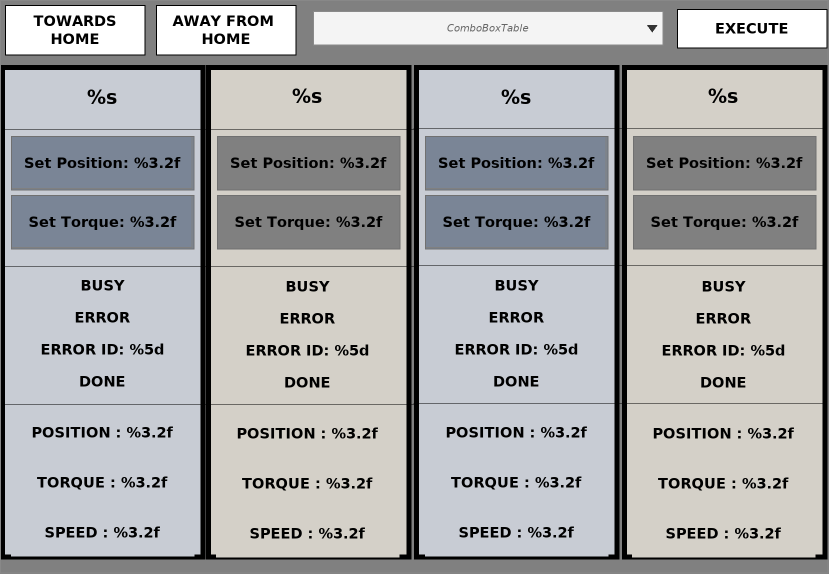
VISUALIZATION motorControlScreen  // 829x574
    Rectangle (206,65 205x494)
    RoundedRectangle (677,9 150x39), "EXECUTE", colour toggle: multiControl.bExecute
        toggle multiControl.bExecute
    ComboBoxTable (313,11 350x34), variable: multiControl.nActionIndex, data array: multiControl.aActionList
        p3854506369: multiControl.aActionList[INDEX]
    Rectangle (0,65 205x494)
    Rectangle (414,65 205x494)
    Rectangle (622,65 205x494)
    RoundedRectangle (10,71 185x53), "%s", text variable: multiControl.sMotorDisp1, colour toggle: multiControl.aMotorEnable[1]
        p55702900: multiControl.aDispFontColor[1]
        toggle multiControl.aMotorEnable[1]
    Rectangle (11,409 183x47), "POSITION : %3.2f", text variable: multiControl.aMotorPos[1]
    Rectangle (11,271 183x29), "BUSY", colour toggle: multiControl.aMotorBusy[1]
    Rectangle (11,367 183x29), "DONE", colour toggle: multiControl.aMotorDone[1]
    Rectangle (11,303 183x29), "ERROR", colour toggle: multiControl.aMotorError[1]
    Rectangle (11,335 183x29), "ERROR ID: %5d", text variable: multiControl.aMotorErrorId[1]
    Rectangle (11,459 183x47), "TORQUE : %3.2f", text variable: multiControl.aMotorTorque[1]
    Rectangle (11,509 183x47), "SPEED : %3.2f", text variable: multiControl.aMotorSpeed[1]
    Button (11,136 183x54), "Set Position: %3.2f", text variable: multiControl.aMotorSetPos[1]
        OnMouseClick: write the text variable via VisuDialogs.Numpad
    Button (11,195 183x54), "Set Torque: %3.2f", text variable: multiControl.aMotorSetTorq[1]
        OnMouseClick: write the text variable via VisuDialogs.Numpad
    Line (0,129) (827,128)
    Line (1,266) (828,265)
    Line (0,404) (827,403)
    Button (217,195 183x54), "Set Torque: %3.2f", text variable: multiControl.aMotorSetTorq[2]
        OnMouseClick: write the text variable via VisuDialogs.Numpad
    Button (217,136 183x54), "Set Position: %3.2f", text variable: multiControl.aMotorSetPos[2]
        OnMouseClick: write the text variable via VisuDialogs.Numpad
    RoundedRectangle (215,70 185x53), "%s", text variable: multiControl.sMotorDisp2, colour toggle: multiControl.aMotorEnable[2]
        p55702900: multiControl.aDispFontColor[2]
        toggle multiControl.aMotorEnable[2]
    Rectangle (216,272 183x29), "BUSY", colour toggle: multiControl.aMotorBusy[2]
    Rectangle (216,410 183x47), "POSITION : %3.2f", text variable: multiControl.aMotorPos[2]
    Rectangle (216,368 183x29), "DONE", colour toggle: multiControl.aMotorDone[2]
    Rectangle (216,304 183x29), "ERROR", colour toggle: multiControl.aMotorError[2]
    Rectangle (216,336 183x29), "ERROR ID: %5d", text variable: multiControl.aMotorErrorId[2]
    Rectangle (216,460 183x47), "TORQUE : %3.2f", text variable: multiControl.aMotorTorque[2]
    Rectangle (216,510 183x47), "SPEED : %3.2f", text variable: multiControl.aMotorSpeed[2]
    RoundedRectangle (424,71 185x53), "%s", text variable: multiControl.sMotorDisp3, colour toggle: multiControl.aMotorEnable[3], invisible if: multiControl.bHideDispMotor3
        p55702900: multiControl.aDispFontColor[3]
        toggle multiControl.aMotorEnable[3]
    Rectangle (425,409 183x47), "POSITION : %3.2f", text variable: multiControl.aMotorPos[3], invisible if: multiControl.bHideDispMotor3
    Rectangle (425,271 183x29), "BUSY", colour toggle: multiControl.aMotorBusy[3], invisible if: multiControl.bHideDispMotor3
    Rectangle (425,367 183x29), "DONE", colour toggle: multiControl.aMotorDone[3], invisible if: multiControl.bHideDispMotor3
    Rectangle (425,303 183x29), "ERROR", colour toggle: multiControl.aMotorError[3], invisible if: multiControl.bHideDispMotor3
    Rectangle (425,335 183x29), "ERROR ID: %5d", text variable: multiControl.aMotorErrorId[3], invisible if: multiControl.bHideDispMotor3
    Rectangle (425,459 183x47), "TORQUE : %3.2f", text variable: multiControl.aMotorTorque[3], invisible if: multiControl.bHideDispMotor3
    Rectangle (425,509 183x47), "SPEED : %3.2f", text variable: multiControl.aMotorSpeed[3], invisible if: multiControl.bHideDispMotor3
    Button (425,136 183x54), "Set Position: %3.2f", text variable: multiControl.aMotorSetPos[3], invisible if: multiControl.bHideDispMotor3
        OnMouseClick: write the text variable via VisuDialogs.Numpad
    Button (425,195 183x54), "Set Torque: %3.2f", text variable: multiControl.aMotorSetTorq[3], invisible if: multiControl.bHideDispMotor3
        OnMouseClick: write the text variable via VisuDialogs.Numpad
    RoundedRectangle (631,70 185x53), "%s", text variable: multiControl.sMotorDisp4, colour toggle: multiControl.aMotorEnable[4], invisible if: multiControl.bHideDispMotor4
        p55702900: multiControl.aDispFontColor[4]
        toggle multiControl.aMotorEnable[4]
    Button (633,195 183x54), "Set Torque: %3.2f", text variable: multiControl.aMotorSetTorq[4], invisible if: multiControl.bHideDispMotor4
        OnMouseClick: write the text variable via VisuDialogs.Numpad
    Button (633,136 183x54), "Set Position: %3.2f", text variable: multiControl.aMotorSetPos[4], invisible if: multiControl.bHideDispMotor4
        OnMouseClick: write the text variable via VisuDialogs.Numpad
    Rectangle (632,272 183x29), "BUSY", colour toggle: multiControl.aMotorBusy[4], invisible if: multiControl.bHideDispMotor4
    Rectangle (632,410 183x47), "POSITION : %3.2f", text variable: multiControl.aMotorPos[4], invisible if: multiControl.bHideDispMotor4
    Rectangle (632,368 183x29), "DONE", colour toggle: multiControl.aMotorDone[4], invisible if: multiControl.bHideDispMotor4
    Rectangle (632,304 183x29), "ERROR", colour toggle: multiControl.aMotorError[4], invisible if: multiControl.bHideDispMotor4
    Rectangle (632,336 183x29), "ERROR ID: %5d", text variable: multiControl.aMotorErrorId[4], invisible if: multiControl.bHideDispMotor4
    Rectangle (632,460 183x47), "TORQUE : %3.2f", text variable: multiControl.aMotorTorque[4], invisible if: multiControl.bHideDispMotor4
    Rectangle (632,510 183x47), "SPEED : %3.2f", text variable: multiControl.aMotorSpeed[4], invisible if: multiControl.bHideDispMotor4
    RoundedRectangle (5,5 140x50), "TOWARDS HOME", colour toggle: multiControl.bHomeDirection, invisible if: multiControl.bHideDirection
        toggle multiControl.bHomeDirection
    RoundedRectangle (156,5 140x50), "AWAY FROM HOME", colour toggle: NOT multiControl.bHomeDirection, invisible if: multiControl.bHideDirection
        toggle multiControl.bHomeDirection
END_VISUALIZATION

(* stored: Version 1.1.0.1, ProductVersion 3.1.4024.13
   Visu motorControlScreen: Id {23ee9f99-c9f3-430a-b145-2f31b2efb83b} *)
